  def rq_is_motion_complete(slave_id):
      detection_flag = driver_gripper_client.getObjectDetectionFlag(slave_id)
      return detection_flag > 0 and detection_flag < 4
  end

  def write_error_popup(slave_id, message_part_1, message_part_2, title):
      popup_message_part_1 = str_cat(message_part_1, rq_slave_id_to_gripper_id(slave_id))
      popup_message_part_2 = str_cat(popup_message_part_1, " ")
      popup_message = str_cat(popup_message_part_2, message_part_2)
      return popup(popup_message, title, False, True, True)
  end

  def rq_slave_id_to_gripper_id(slave_id):
      if slave_id == 9:
          return 1
      else:
          return slave_id
      end
  end

  def rq_disconnect_grippers():
      driver_gripper_client.pauseAndDisconnect()
  end

  def rq_reconnect_grippers(blocking=False, slave_ids=[], halt_on_error=True):
      if blocking:
          gripper_reconnecting = True
          local reconnection_success = driver_gripper_client.reconnectAndResume(slave_ids)
          gripper_reconnecting = False

          if (not reconnection_success and halt_on_error):
            popup("Could not reconnect to grippers", error=True)
            halt
          else:
            return reconnection_success
          end
      else:
          thread recon_thread():
              rq_reconnect_grippers(True)
              return False
          end
          thrd = run recon_thread()
      end
  end

  def rq_wait_for_gripper_reconnection(timeout_s = 30.0):
      while (gripper_reconnecting == True):
          if (timeout_s <= 0):
            popup("Gripper has not reconnected before the expected time")
            halt
          else:
            sync()
            timeout_s = timeout_s - get_steptime()
          end
      end
  end

  def rq_gripper_allow_tool_com(allow_tool_comm):
      driver_gripper_client.allowToolComm(allow_tool_comm)
  end
  set_closed_norm(100.0, "1")
  set_open_norm(0.0, "1")
  set_closed_mm(0.0, "1")
  set_open_mm(50.0, "1")
  set_closed_norm(100.0, "2")
  set_open_norm(0.0, "2")
  set_closed_mm(0.0, "2")
  set_open_mm(50.0, "2")
  set_closed_norm(100.0, "3")
  set_open_norm(0.0, "3")
  set_closed_mm(0.0, "3")
  set_open_mm(50.0, "3")
  set_closed_norm(100.0, "4")
  set_open_norm(0.0, "4")
  set_closed_mm(0.0, "4")
  set_open_mm(50.0, "4")
  rq_current_limit_enabled = False
  # end: URCap Installation Node
  step_count_fc6ca3d9_0ff9_45fd_874f_89cc75eebf0e = 0.0
  thread Step_Counter_Thread_1f0c7b0e_410d_4908_aa3c_46b36282060a():
    while (True):
      step_count_fc6ca3d9_0ff9_45fd_874f_89cc75eebf0e = step_count_fc6ca3d9_0ff9_45fd_874f_89cc75eebf0e + 1.0
      sync()
    end
  end
  run Step_Counter_Thread_1f0c7b0e_410d_4908_aa3c_46b36282060a()
  while (True):
    $ 2 "로봇 프로그램"
    # begin: URCap Program Node
    #   Source: Robotiq_Grippers, 3.27.0.122343, Robotiq Inc.
    #   Type: 그립퍼 활성화
    $ 3 "그립퍼 활성화"

    rq_set_max_current_for_all_grippers()

    reset_and_activate = False

    rq_activate_all_grippers(False)
    # end: URCap Program Node
    $ 4 "5회 Loop:"
    u47336u54532_1 = 0
    while (u47336u54532_1 < 5):
      # begin: URCap Program Node
      #   Source: OnRobot, 5.14.3, OnRobot A/S
      #   Type: 2FG 그립
      $ 5 "2FG 그립 (33)"
on_return = twofg_grip(width=33.0, force=50, speed=100, external_grip=True, tool_index=0)
twofg_payload_set(mass = 0.0, tool_index = 0, use_guard = True)
      # end: URCap Program Node
      # begin: URCap Program Node
      #   Source: OnRobot, 5.14.3, OnRobot A/S
      #   Type: 2FG 놓기
      $ 6 "2FG 놓기 (70)"
on_return = twofg_release(width=70.0, speed=100, external_release=True, tool_index=0 )
twofg_payload_set(mass = 0.0, tool_index = 0, use_guard = False)
      # end: URCap Program Node
      u47336u54532_1 = u47336u54532_1 + 1
    end
  end
end
